TYPE U_INSTANCE_STATE :
UNION
  stState             : ARRAY[1..MAX_PROCESS] OF ST_INSTANCE_STATE;
  byState   AT %Q*    : ARRAY[1..MAX_PROCESS] OF
                        ARRAY[1..SIZEOF(ST_INSTANCE_STATE)] OF BYTE;
END_UNION
END_TYPE

(* stored: Version 1.1.0.1, ProductVersion 3.1.4026.13
   DUT U_INSTANCE_STATE: Id {dab65295-5f94-4c03-a860-8c1f4f040107} *)
